TYPE ST_Enclosure_get :
STRUCT
	climate				: ST_EnclosureClimate_Get;
	doors				: ST_DoorsNLocks_get;
	ledstrip			: ST_Ledstrip_get;
END_STRUCT
END_TYPE

(* stored: Version 1.1.0.1, ProductVersion 3.1.4026.18
   DUT ST_Enclosure_get: Id {a884b94b-5278-45e4-8e11-5ffcd334137c} *)
